# EPICS substitutions: iocBoot/ioc13MeasCompE1608_1/pid_slow.substitutions
file "$(STD)/stdApp/Db/pid_control.db"
{
pattern
{P,            PID,        INP,    OUT,         LOPR,  HOPR,  DRVL,  DRVH,  PREC,   KP,  KI,   KD,  SCAN}
{13E1608_1:, PID1, 13ETC_1:Ti0,  13E1608_1:Ao1,   0,    10,     0,    10,     3,    1.2,  1.,   0.,  ".1 second"}
}
